PROGRAM q_Gestion_Actionneurs_ANA
VAR
	Moteur_Aerobox_Bas_Deb: Moteur_EC;
	Batterie_Electrique: BatElec;
	Moteur_By_Pass: Moteur_EC;
	Reg_Etanche_Ext: Registre_V1;
	V3V_Eau_Mitig: Registre_V1;
END_VAR
VAR // added by the converter: edge detectors and wires of the graphical bodies
    _w1 : BOOL;
END_VAR

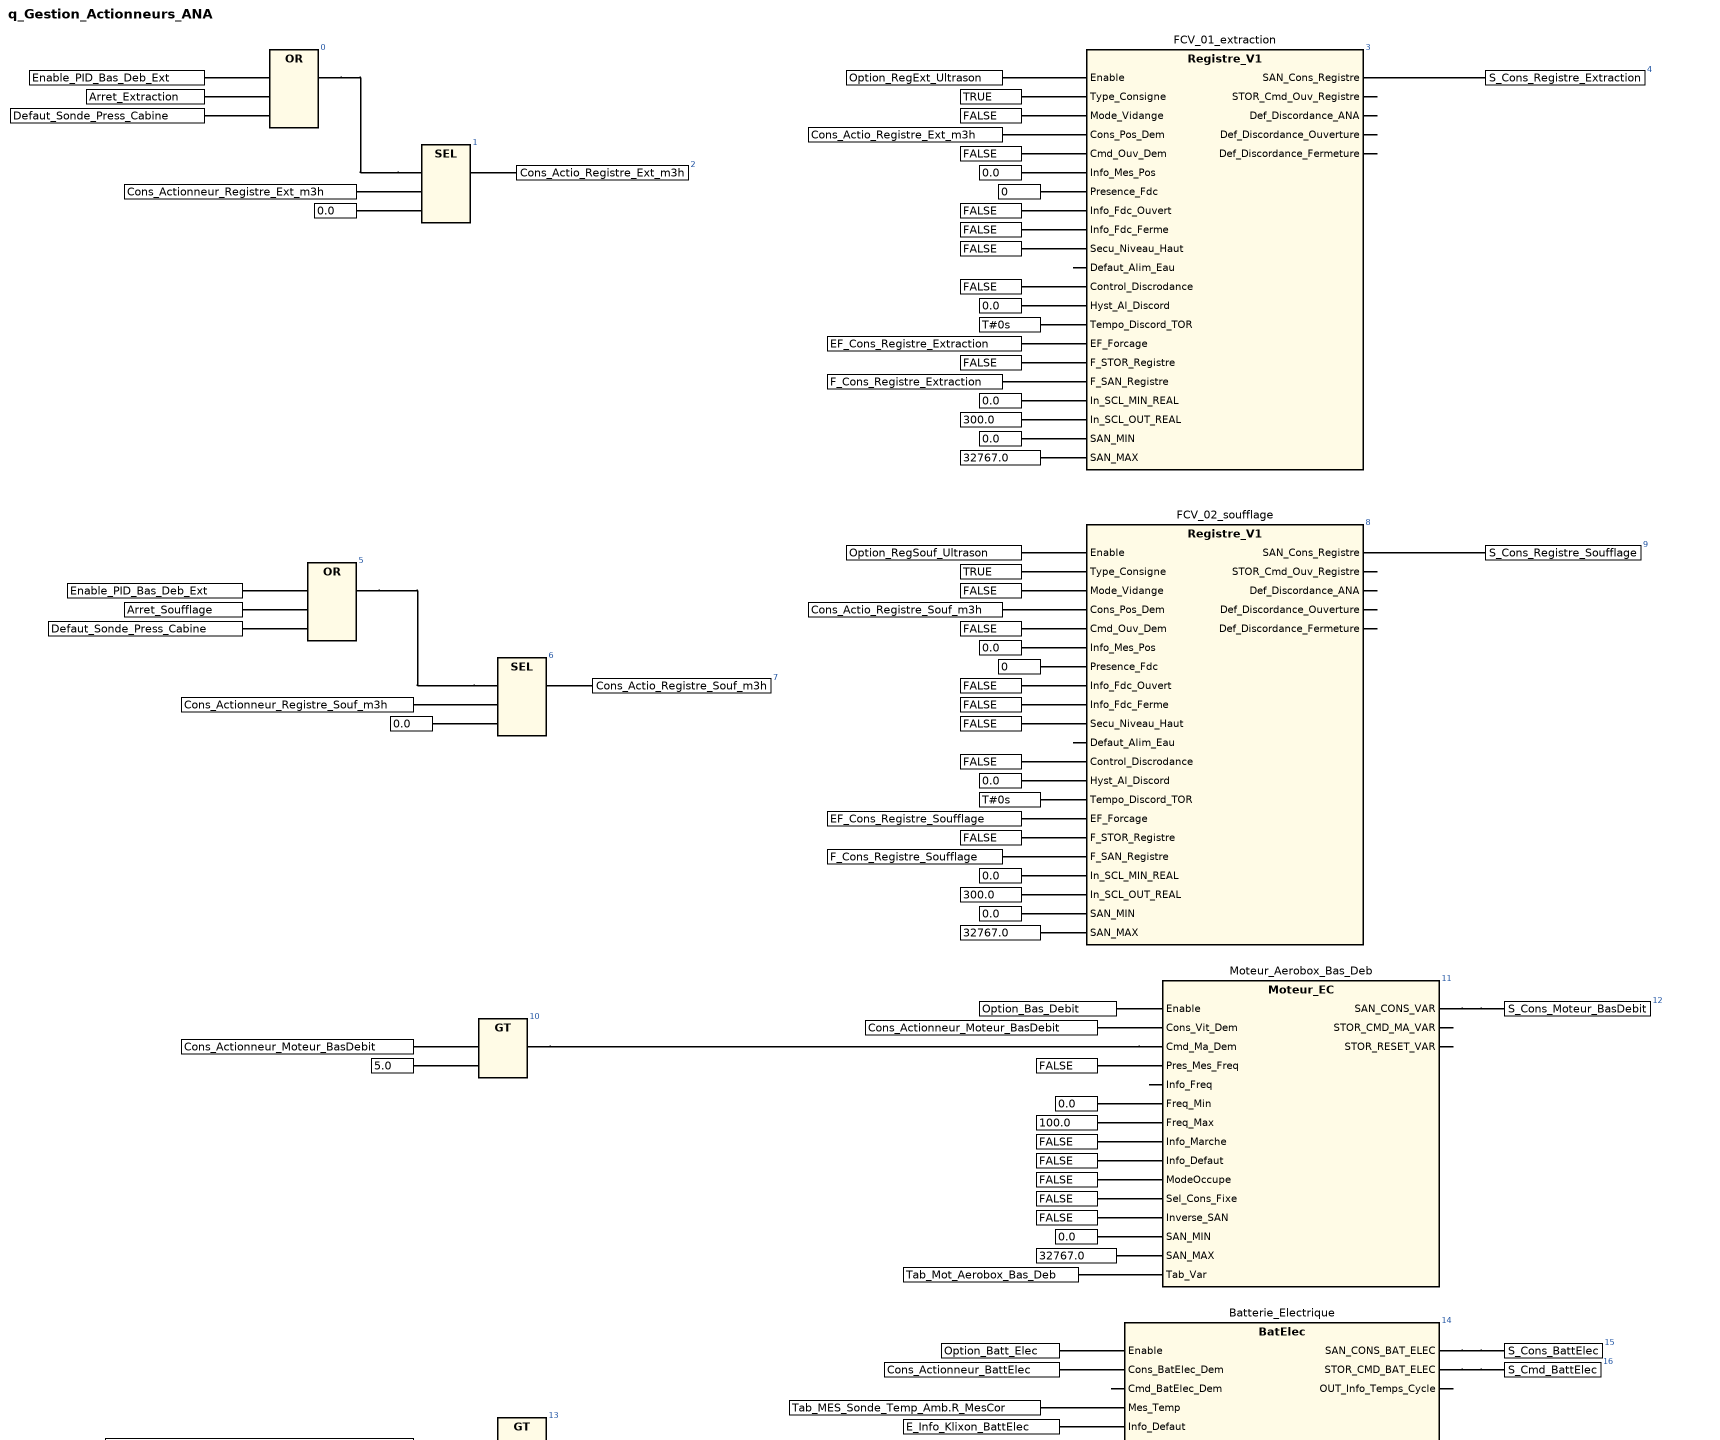
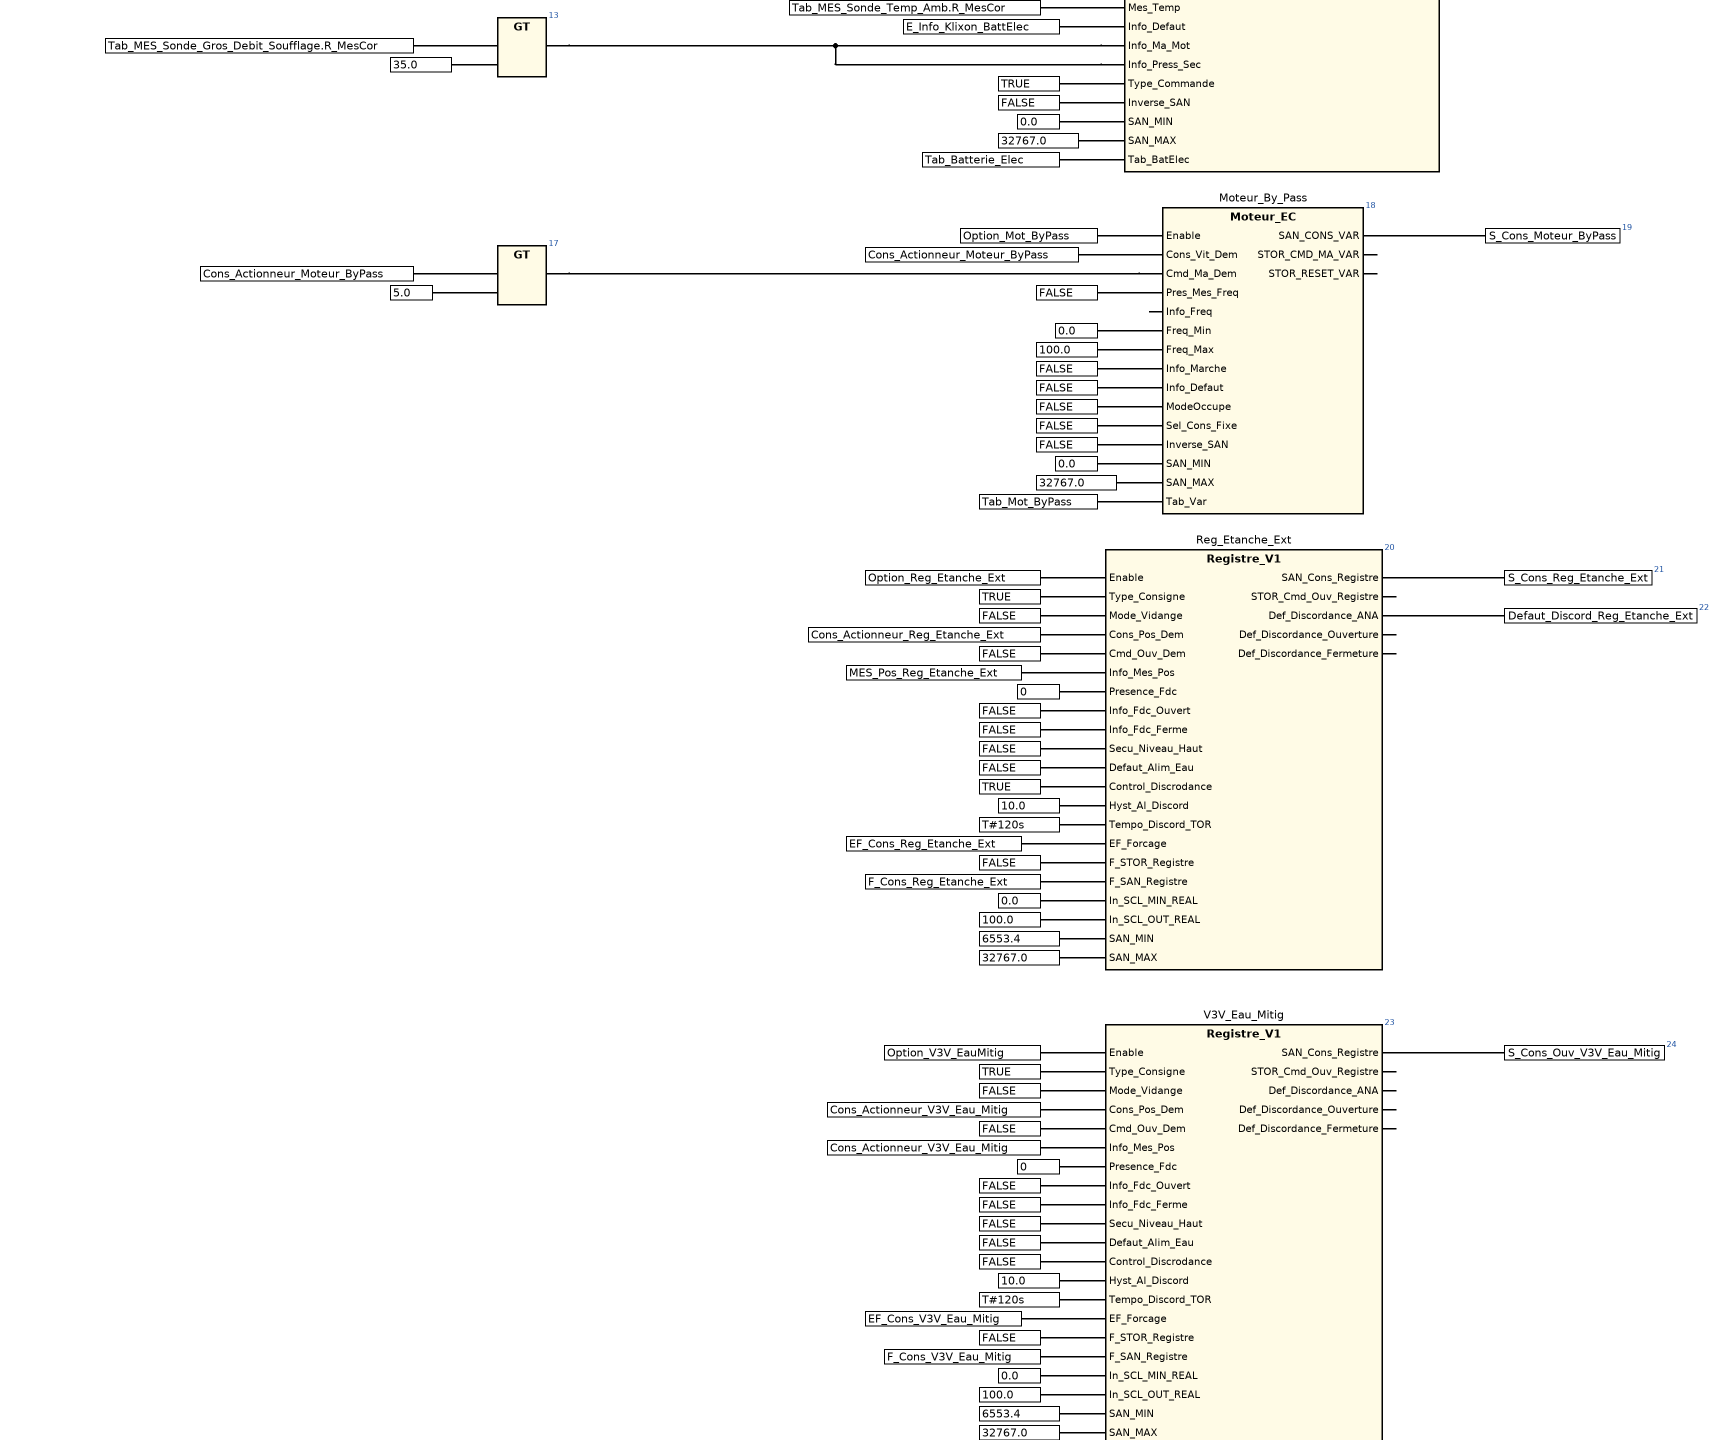
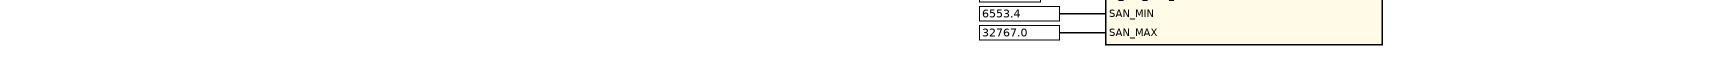
Cons_Actio_Registre_Ext_m3h := SEL(Enable_PID_Bas_Deb_Ext OR Arret_Extraction OR Defaut_Sonde_Press_Cabine, Cons_Actionneur_Registre_Ext_m3h, 0.0);
FCV_01_extraction(
    Enable := Option_RegExt_Ultrason,
    Type_Consigne := TRUE,
    Mode_Vidange := FALSE,
    Cons_Pos_Dem := Cons_Actio_Registre_Ext_m3h,
    Cmd_Ouv_Dem := FALSE,
    Info_Mes_Pos := 0.0,
    Presence_Fdc := 0,
    Info_Fdc_Ouvert := FALSE,
    Info_Fdc_Ferme := FALSE,
    Secu_Niveau_Haut := FALSE,
    Control_Discrodance := FALSE,
    Hyst_Al_Discord := 0.0,
    Tempo_Discord_TOR := T#0s,
    EF_Forcage := EF_Cons_Registre_Extraction,
    F_STOR_Registre := FALSE,
    F_SAN_Registre := F_Cons_Registre_Extraction,
    In_SCL_MIN_REAL := 0.0,
    In_SCL_OUT_REAL := 300.0,
    SAN_MIN := 0.0,
    SAN_MAX := 32767.0); // Registre_V1
S_Cons_Registre_Extraction := FCV_01_extraction.SAN_Cons_Registre;
Cons_Actio_Registre_Souf_m3h := SEL(Enable_PID_Bas_Deb_Ext OR Arret_Soufflage OR Defaut_Sonde_Press_Cabine, Cons_Actionneur_Registre_Souf_m3h, 0.0);
FCV_02_soufflage(
    Enable := Option_RegSouf_Ultrason,
    Type_Consigne := TRUE,
    Mode_Vidange := FALSE,
    Cons_Pos_Dem := Cons_Actio_Registre_Souf_m3h,
    Cmd_Ouv_Dem := FALSE,
    Info_Mes_Pos := 0.0,
    Presence_Fdc := 0,
    Info_Fdc_Ouvert := FALSE,
    Info_Fdc_Ferme := FALSE,
    Secu_Niveau_Haut := FALSE,
    Control_Discrodance := FALSE,
    Hyst_Al_Discord := 0.0,
    Tempo_Discord_TOR := T#0s,
    EF_Forcage := EF_Cons_Registre_Soufflage,
    F_STOR_Registre := FALSE,
    F_SAN_Registre := F_Cons_Registre_Soufflage,
    In_SCL_MIN_REAL := 0.0,
    In_SCL_OUT_REAL := 300.0,
    SAN_MIN := 0.0,
    SAN_MAX := 32767.0); // Registre_V1
S_Cons_Registre_Soufflage := FCV_02_soufflage.SAN_Cons_Registre;
Moteur_Aerobox_Bas_Deb(
    Enable := Option_Bas_Debit,
    Cons_Vit_Dem := Cons_Actionneur_Moteur_BasDebit,
    Cmd_Ma_Dem := Cons_Actionneur_Moteur_BasDebit > 5.0,
    Pres_Mes_Freq := FALSE,
    Freq_Min := 0.0,
    Freq_Max := 100.0,
    Info_Marche := FALSE,
    Info_Defaut := FALSE,
    ModeOccupe := FALSE,
    Sel_Cons_Fixe := FALSE,
    Inverse_SAN := FALSE,
    SAN_MIN := 0.0,
    SAN_MAX := 32767.0,
    Tab_Var := Tab_Mot_Aerobox_Bas_Deb); // Moteur_EC
S_Cons_Moteur_BasDebit := Moteur_Aerobox_Bas_Deb.SAN_CONS_VAR;
_w1 := Tab_MES_Sonde_Gros_Debit_Soufflage.R_MesCor > 35.0;
Batterie_Electrique(
    Enable := Option_Batt_Elec,
    Cons_BatElec_Dem := Cons_Actionneur_BattElec,
    Mes_Temp := Tab_MES_Sonde_Temp_Amb.R_MesCor,
    Info_Defaut := E_Info_Klixon_BattElec,
    Info_Ma_Mot := _w1,
    Info_Press_Sec := _w1,
    Type_Commande := TRUE,
    Inverse_SAN := FALSE,
    SAN_MIN := 0.0,
    SAN_MAX := 32767.0,
    Tab_BatElec := Tab_Batterie_Elec); // BatElec
S_Cons_BattElec := Batterie_Electrique.SAN_CONS_BAT_ELEC;
S_Cmd_BattElec := Batterie_Electrique.STOR_CMD_BAT_ELEC;
Moteur_By_Pass(
    Enable := Option_Mot_ByPass,
    Cons_Vit_Dem := Cons_Actionneur_Moteur_ByPass,
    Cmd_Ma_Dem := Cons_Actionneur_Moteur_ByPass > 5.0,
    Pres_Mes_Freq := FALSE,
    Freq_Min := 0.0,
    Freq_Max := 100.0,
    Info_Marche := FALSE,
    Info_Defaut := FALSE,
    ModeOccupe := FALSE,
    Sel_Cons_Fixe := FALSE,
    Inverse_SAN := FALSE,
    SAN_MIN := 0.0,
    SAN_MAX := 32767.0,
    Tab_Var := Tab_Mot_ByPass); // Moteur_EC
S_Cons_Moteur_ByPass := Moteur_By_Pass.SAN_CONS_VAR;
Reg_Etanche_Ext(
    Enable := Option_Reg_Etanche_Ext,
    Type_Consigne := TRUE,
    Mode_Vidange := FALSE,
    Cons_Pos_Dem := Cons_Actionneur_Reg_Etanche_Ext,
    Cmd_Ouv_Dem := FALSE,
    Info_Mes_Pos := MES_Pos_Reg_Etanche_Ext,
    Presence_Fdc := 0,
    Info_Fdc_Ouvert := FALSE,
    Info_Fdc_Ferme := FALSE,
    Secu_Niveau_Haut := FALSE,
    Defaut_Alim_Eau := FALSE,
    Control_Discrodance := TRUE,
    Hyst_Al_Discord := 10.0,
    Tempo_Discord_TOR := T#120s,
    EF_Forcage := EF_Cons_Reg_Etanche_Ext,
    F_STOR_Registre := FALSE,
    F_SAN_Registre := F_Cons_Reg_Etanche_Ext,
    In_SCL_MIN_REAL := 0.0,
    In_SCL_OUT_REAL := 100.0,
    SAN_MIN := 6553.4,
    SAN_MAX := 32767.0); // Registre_V1
S_Cons_Reg_Etanche_Ext := Reg_Etanche_Ext.SAN_Cons_Registre;
Defaut_Discord_Reg_Etanche_Ext := Reg_Etanche_Ext.Def_Discordance_ANA;
V3V_Eau_Mitig(
    Enable := Option_V3V_EauMitig,
    Type_Consigne := TRUE,
    Mode_Vidange := FALSE,
    Cons_Pos_Dem := Cons_Actionneur_V3V_Eau_Mitig,
    Cmd_Ouv_Dem := FALSE,
    Info_Mes_Pos := Cons_Actionneur_V3V_Eau_Mitig,
    Presence_Fdc := 0,
    Info_Fdc_Ouvert := FALSE,
    Info_Fdc_Ferme := FALSE,
    Secu_Niveau_Haut := FALSE,
    Defaut_Alim_Eau := FALSE,
    Control_Discrodance := FALSE,
    Hyst_Al_Discord := 10.0,
    Tempo_Discord_TOR := T#120s,
    EF_Forcage := EF_Cons_V3V_Eau_Mitig,
    F_STOR_Registre := FALSE,
    F_SAN_Registre := F_Cons_V3V_Eau_Mitig,
    In_SCL_MIN_REAL := 0.0,
    In_SCL_OUT_REAL := 100.0,
    SAN_MIN := 6553.4,
    SAN_MAX := 32767.0); // Registre_V1
S_Cons_Ouv_V3V_Eau_Mitig := V3V_Eau_Mitig.SAN_Cons_Registre;

END_PROGRAM

(* stored: Version 1.1.0.1, ProductVersion 3.1.4024.12
   POU q_Gestion_Actionneurs_ANA: Id {b7e99b63-f4e6-4821-9f8d-75adca4b868c}, SpecialFunc None *)
